Fanuc KAREL source: kt00728.KL

PROGRAM KT00728
%STACKSIZE=65535
%PRIORITY=65535
%NOLOCKGROUP
VAR
OUT : BOOLEAN
-- UNRESOLVED DECLARATIONS (source type spelling not recovered)
-- C1 : TYPE_0x001C (type_u16=0x001C)
-- C2 : TYPE_0x001C (type_u16=0x001C)
BEGIN
-- UNRESOLVED_PC line 8 opcodes [9D 22 A5] marker_code=0
-- UNRESOLVED_PC line 9 opcodes [9C 22 A5] marker_code=15
-- UNRESOLVED_PC line 10 opcodes [9D 22 A5] marker_code=30
-- UNRESOLVED_PC line 11 opcodes [9C 22 A5] marker_code=45
-- UNRESOLVED_PC line 12 opcodes [22 63 23] marker_code=60
END KT00728
